FUNCTION F_Int2Real : REAL
VAR_INPUT
	nIn: INT;
	nDecimal: INT;
END_VAR
VAR
	rVal: REAL;
END_VAR

rVal:= INT_TO_REAL(nIn);	
CASE nDecimal OF
	1:  
		rVal := rVal / 10;
	2:     
		rVal := rVal / 100;
	3:
		rVal := rVal / 1000;    
END_CASE;
F_Int2Real := rVal;

END_FUNCTION

(* stored: Version 1.1.0.1, ProductVersion 3.1.4024.12
   POU F_Int2Real: Id {a83141dd-c5bc-4ba9-a29a-a1ffe92daa2e}, SpecialFunc None *)
